// TIA Portal V16 export
// export: Created 2024-12-03T15:41:41.3205342Z, ExportSetting WithDefaults, DisplayName Totally Integrated Automation Portal, DisplayVersion V16 Update 6, DisplayName TIA Portal Version Control Interface, DisplayVersion V16 Update 2, DisplayName TIA Portal Openness, DisplayVersion V16 Update 6, DisplayName TIA Portal Teamcenter Gateway, DisplayVersion V16, DisplayName SINAMICS Startdrive Advanced, DisplayVersion V16 Update 5, DisplayName SINAMICS Startdrive G130, G150, S120, S150, SINAMICS MV, S210, DisplayVersion V16 Update 5, DisplayName SINAMICS Startdrive G110M, G120, G120C, G120D, G120P, G115D, DisplayVersion V16 Update 5, DisplayName STEP 7 Professional, DisplayVersion V16 Update 6, DisplayName STEP 7 Safety, DisplayVersion V16, DisplayName WinCC Advanced / Unified PC, DisplayVersion V16 Update 6
FUNCTION_BLOCK "TOFF_Encoder_FB"   // FB57, SCL
{ S7_Optimized_Access := 'TRUE' }
VERSION : 0.1
// stored: AutoNumber true, IsIECCheckEnabled false, IsRetainMemResEnabled false, MemoryReserve 100, SetENOAutomatically false, UDAEnableTagReadback false
   VAR_INPUT
      I_DeltaDistance_mm : Real;   // The distance traveld mm / PLC cycle
      I_SetPoint : Real;   // Preset value
      I_Start : Bool;   // Start counting the distance
      I_Reset : Bool;   // Reset distance
      I_ResetHandshake : Bool;
   END_VAR
   VAR_OUTPUT
      Q : Bool;   // Distance is traveld
   END_VAR
   VAR
      StartCount : Bool;
      signal : "SmartBool";
      DistanceMem : Real;
   END_VAR
BEGIN
   #signal(I_Sensor:= #I_Start);

   IF #signal.O_data.FE THEN
       #StartCount := true;
   END_IF;

   IF #signal.O_data.State THEN
       #DistanceMem := 0.0;
       #StartCount := FALSE;
   END_IF;

   IF #StartCount AND #DistanceMem < #I_SetPoint THEN
       #DistanceMem += #I_DeltaDistance_mm;
   END_IF;

   IF #DistanceMem >= #I_SetPoint THEN
       #StartCount := 0;
       #DistanceMem := 0.0;
   END_IF;

   IF #I_Reset OR #I_ResetHandshake THEN
       #StartCount := FALSE;
       #DistanceMem := 0.0;
   END_IF;

   #Q := #StartCount OR #I_Start;

   IF #I_ResetHandshake THEN
       #I_ResetHandshake := 0;
   END_IF;
END_FUNCTION_BLOCK
